Staubli VAL3: delete.pgx

public program delete(num x_nIndexTool)
begin
  delete(saveData:tData[x_nIndexTool])
end
